{attribute 'qualified_only'}
VAR_GLOBAL
	PrintingBed		: ST_PrintingBed;
END_VAR

(* stored: Version 1.1.0.1
   GVL GVL_PrintingBed: Id {ccb70eb2-a468-4628-ae77-1cc016a63a53} *)
